RoboDK station: Test-Comau.rdk

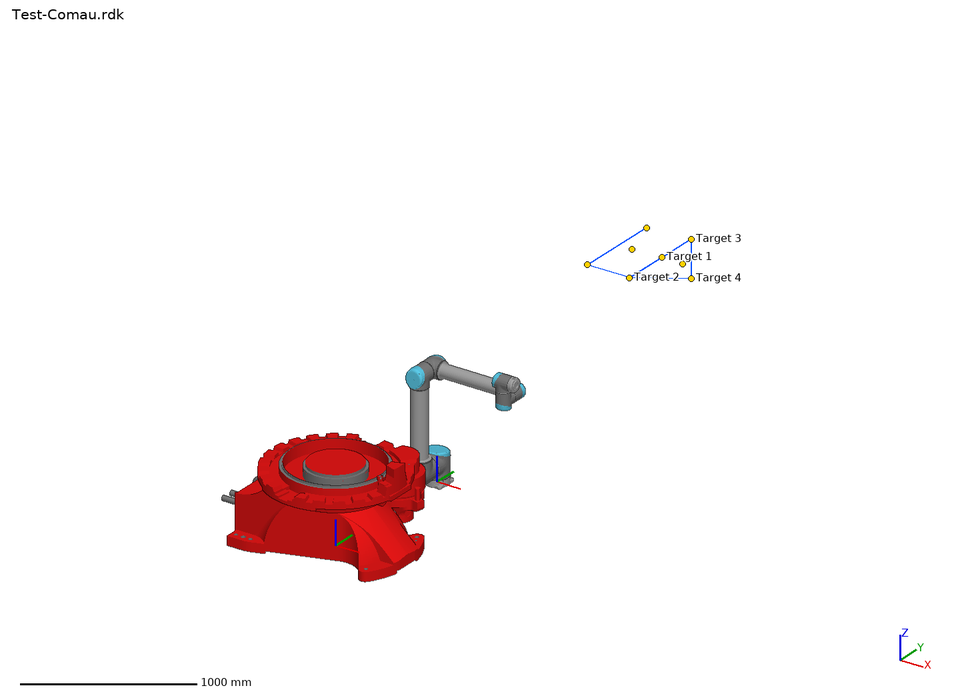
[picture v0: the station drawn from its stored meshes, robots at their saved joint values, targets as dots, program paths as lines]
Station Test-Comau. Poses are relative to the parent item; angles as X-Y-Z fixed-axis rotations.
Station parameters (name, value as stored): IO_5, 1
  - frame Comau NJ 370-3.0 Base at (0, 0, 0) mm
    - robot Comau NJ 370-3.0: 6 axes, payload 370 kg, reach 1436 mm, repeatability 0.15 mm, weight 2450 kg
        joint limits [-180, -60, -231, -400, -125, -720] to [180, 75, -10, 400, 125, 720]; home [0, 0, -90, 0, 0, 0]; saved at [10.766, -14.127, -88.793, -83.678, 10.833, 83.564]
      - tool Tool, TCP at (0, 0, 0) mm
    - target Target 1 (Cartesian target) at (2252, 0, 2440) mm, rotated rx 0 ry 90 rz 0 deg; joints [0, 0, -90, 0, 0, 0] of Comau NJ 370-3.0
    - target Target 2 (Cartesian target) at (2252, -319.08, 2440) mm, rotated rx 0 ry 90 rz 0 deg; joints [9.2, 1.404, -89.988, -89.926, 9.2, 89.925] of Comau NJ 370-3.0
    - target Target 3 (Cartesian target) at (2252, 288.21, 2440) mm, rotated rx 0 ry 90 rz 0 deg; joints [-8.323, 1.146, -89.992, -90.054, -8.323, 90.055] of Comau NJ 370-3.0
    - target Target 4 (Cartesian target) at (2252, 288.21, 2191.35) mm, rotated rx 0 ry 90 rz 0 deg; joints [-8.323, 0.023, -99.35, -42.002, -12.493, 41.32] of Comau NJ 370-3.0
    - target Target 5 (Cartesian target) at (2393.31, 0, 2440) mm, rotated rx 0 ry 90 rz 0 deg; joints [0, 7.825, -89.629, 0, 0.371, 0] of Comau NJ 370-3.0
    - target Target 6 (Cartesian target) at (1960.05, -319.08, 2440) mm, rotated rx 0 ry 90 rz 0 deg; joints [10.766, -14.127, -88.793, -83.678, 10.833, 83.564] of Comau NJ 370-3.0
    - target Target 7 (Cartesian target) at (1960.05, 265.51, 2440) mm, rotated rx 0 ry 90 rz 0 deg; joints [-8.991, -14.621, -88.707, 81.885, 9.083, -81.783] of Comau NJ 370-3.0
    - target Target 8 (Cartesian target) at (2050.36, -10.65, 2440) mm, rotated rx 0 ry 90 rz 0 deg; joints [0.345, -10.889, -89.282, -25.662, 0.797, 25.66] of Comau NJ 370-3.0
  - program Prog1 (15 instructions, listed below)
  - frame UR10 Base at (0, 1000, 0) mm
    - robot UR10: 6 axes, payload 10 kg, reach 1300 mm, repeatability 0.1 mm, weight 28.9 kg
        modified DH rows (alpha deg, a mm, theta deg, d mm): 0, 0, 0, 128; 90, 0, 180, 0; 0, 612.7, 0, 0; 0, 571.6, 0, 163.9; -90, 0, 0, 115.7; 90, 0, 180, 92.2
        joint limits [-360, -360, -360, -360, -360, -360] to [360, 360, 360, 360, 360, 360]; home [0, -90, -90, 0, 90, 0]; saved at [0, -90, -90, 0, 90, 0]
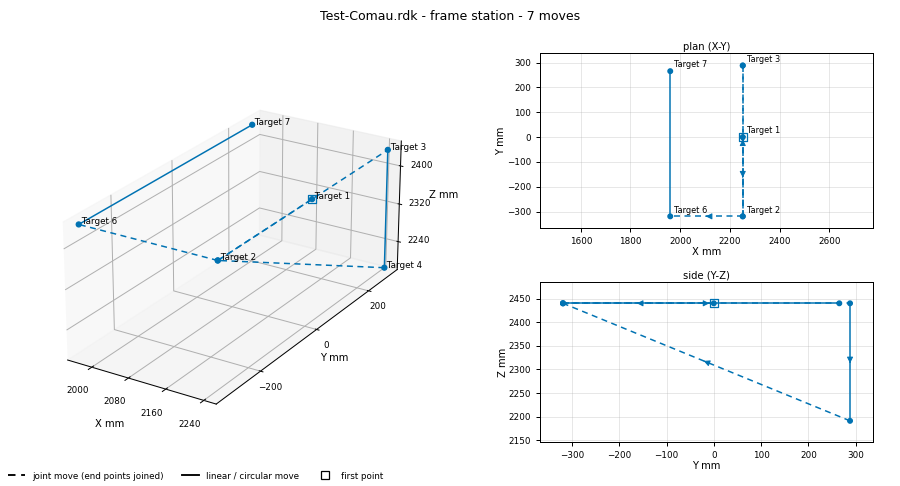
[picture p0: tool path of Test-Comau.rdk in frame station, 7 of 7 moves have a stored position in this frame; points joined in program order, loops and branches not executed]

--- program Prog1 (robot Comau NJ 370-3.0) ---
  Set Ref.: Comau NJ 370-3.0 Base
  MoveJ (Target 1)
  MoveJ (Target 2)
  MoveJ (Target 3)
  MoveL (Target 4)
  MoveJ (Target 2)
  MoveJ (Target 6)
  MoveC (Target 6, Target 7)
  Print: Display message
  Call Program1
  Set IO_5=1
  Wait IO_5=1 T5.0s
  Set Ref.: Comau NJ 370-3.0 Base
  Set Tool
  Set speed (500.0 mm/s)
